FUNCTION_BLOCK EBSlave2301 (* Service Interface Function Block Type *)
  (* Description: Copyright (c) 2016 fortiss GmbH This program and the accompanying materials are made available under the terms of the Eclipse Public License 2.0 which is available at https://www.eclipse.org/legal/epl-2.0/ SPDX-License-Identifier: EPL-2.0 *)
  (* Version 1.0, 2016-11-30, Johannes Messmer, fortiss GmbH *)
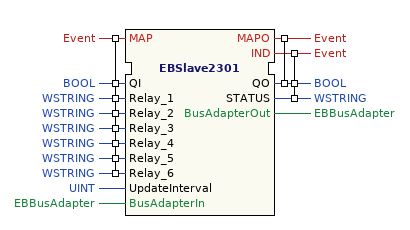
  EVENT_INPUT
    MAP WITH Relay_1, Relay_2, Relay_3, Relay_4, Relay_5, Relay_6, QI; (* Map Pins *)
  END_EVENT
  EVENT_OUTPUT
    MAPO WITH QO; (* Confirm Pin Mapping *)
    IND WITH QO, STATUS; (* Indication from Resource *)
  END_EVENT
  VAR_INPUT
    QI : BOOL; (* Event Input Qualifier *)
    Relay_1 : WSTRING;
    Relay_2 : WSTRING;
    Relay_3 : WSTRING;
    Relay_4 : WSTRING;
    Relay_5 : WSTRING;
    Relay_6 : WSTRING;
    UpdateInterval : UINT; (* Update interval of slave module in Hz (inherited from Master) *)
  END_VAR
  VAR_OUTPUT
    QO : BOOL; (* Event Output Qualifier *)
    STATUS : WSTRING; (* Service Status *)
  END_VAR
  SOCKETS
    BusAdapterIn : EBBusAdapter;
  END_SOCKETS
  PLUGS
    BusAdapterOut : EBBusAdapter;
  END_PLUGS
END_FUNCTION_BLOCK
